// TIA Portal V20 program export: 1 tag tables, 1 data types, 3 data blocks, 8 code blocks (in call order from the OBs), 3 instance data blocks

VAR_GLOBAL   // PLC tag table "Default tag table"
   Tag_1 AT %M1.0 : Bool;
   Tag_2 AT %M10.0 : Bool;
   Tag_3 AT %M10.1 : Bool;
   Tag_4 AT %M10.2 : Bool;
   Tag_5 AT %M10.3 : Bool;
END_VAR

TYPE "F-link_UDT"
// stored: IsFailsafeCompliant true
   STRUCT
      ESTOP_OK : Bool;
      ESTOP_ack_req : Bool;
   END_STRUCT;
END_TYPE

DATA_BLOCK "Adatok_G2"   // DB2
{ S7_Optimized_Access := 'TRUE' }
// stored: MemoryReserve 100
BEGIN
END_DATA_BLOCK

DATA_BLOCK "Data_to_Safety"   // DB3
{ S7_Optimized_Access := 'TRUE' }
// stored: MemoryReserve 100
   VAR
      rcv_buffer : Array[0..121] of Byte;
      rcv_buffer2 : Array[0..121] of Byte;
   END_VAR
BEGIN
END_DATA_BLOCK

DATA_BLOCK "F-link_DB"   // DB2
{ S7_Optimized_Access := 'TRUE' }
// stored: MemoryReserve 100
   VAR
      receive : "F-link_UDT";
   END_VAR
BEGIN
END_DATA_BLOCK

ORGANIZATION_BLOCK "Main"   // OB1, LAD, ProgramCycle
TITLE = "Main Program Sweep (Cycle)"
{ S7_Optimized_Access := 'TRUE' }
// stored: SetENOAutomatically false
   VAR_INPUT
      Initial_Call : Bool;   // Initial call of this OB
      Remanence : Bool;   // =True, if remanent data are available
   END_VAR
BEGIN

REGION Network 1
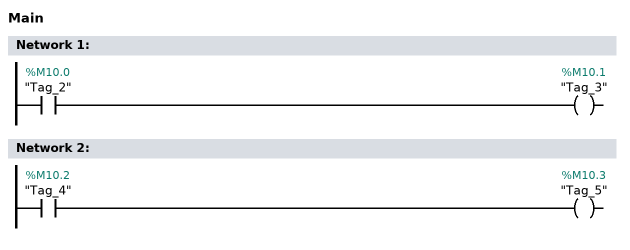
   RUNG wire#powerrail
      Contact( "Tag_2" )
      Coil( "Tag_3" )
   END_RUNG
   // the same network as SCL:
   "Tag_3" := "Tag_2";
END_REGION

REGION Network 2
   RUNG wire#powerrail
      Contact( "Tag_4" )
      Coil( "Tag_5" )
   END_RUNG
   // the same network as SCL:
   "Tag_5" := "Tag_4";
END_REGION
END_ORGANIZATION_BLOCK

ORGANIZATION_BLOCK "CyclicInterrupt"   // OB30, LAD, CyclicInterrupt
{ S7_Optimized_Access := 'TRUE' }
// stored: SetENOAutomatically false
   VAR_INPUT
      Initial_Call : Bool;   // Initial call of this OB
      Event_Count : Int;   // Events discarded
   END_VAR
BEGIN

REGION Network 1
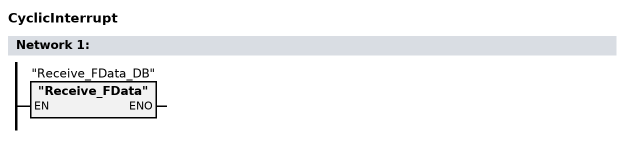
   RUNG wire#powerrail
      "Receive_FData_DB"()
   END_RUNG
   // the same network as SCL:
   "Receive_FData_DB"();   // "Receive_FData"
END_REGION
END_ORGANIZATION_BLOCK

FUNCTION_BLOCK "Receive_FData"   // FB2, FBD
{ S7_Optimized_Access := 'TRUE' }
// stored: MemoryReserve 100, SetENOAutomatically false
   VAR
      TRCV_Instance { S7_SetPoint := 'True'} : TRCV;
   END_VAR
BEGIN

REGION Network 1: ACK tömb fogadása
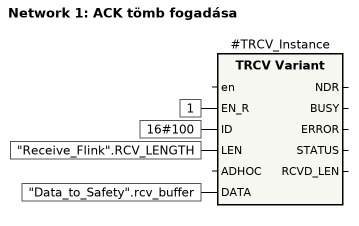
   #TRCV_Instance(EN_R := 1,   // TRCV
                  ID := 16#100,
                  LEN := "Receive_Flink".RCV_LENGTH,
                  DATA := "Data_to_Safety".rcv_buffer);
END_REGION
END_FUNCTION_BLOCK

FUNCTION_BLOCK "Main_Safety_RTG1"   // FB1, F_FBD
{ S7_Optimized_Access := 'TRUE' }
// stored: AutoNumber false
   VAR
      ESTOP1_Instance : ESTOP1;
   END_VAR
BEGIN

REGION Network 1
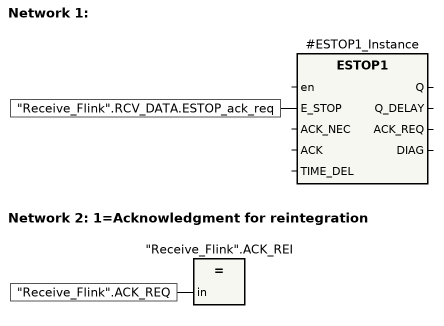
   #ESTOP1_Instance(E_STOP := "Receive_Flink".RCV_DATA.ESTOP_ack_req);   // ESTOP1
END_REGION

REGION Network 2: 1=Acknowledgment for reintegration
   "Receive_Flink".ACK_REI := "Receive_Flink".ACK_REQ;
END_REGION
END_FUNCTION_BLOCK

FUNCTION "PostProcess_Send" : Void   // FC2, FBD
{ S7_Optimized_Access := 'TRUE' }
// stored: SetENOAutomatically false
BEGIN

REGION Network 1
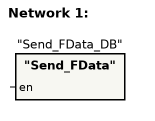
   "Send_FData_DB"();   // "Send_FData"
END_REGION
END_FUNCTION

FUNCTION_BLOCK "Send_FData"   // FB3, FBD
{ S7_Optimized_Access := 'TRUE' }
// stored: MemoryReserve 100, SetENOAutomatically false
   VAR
      TSEND_Instance { S7_SetPoint := 'True'} : TSEND;
      status_save { S7_SetPoint := 'True'} : Word;
      trigger : Bool;
   END_VAR
   VAR_TEMP   // added for the SCL form of the ladder/FBD networks
      _w1 : Bool;
   END_VAR
BEGIN

REGION Network 1
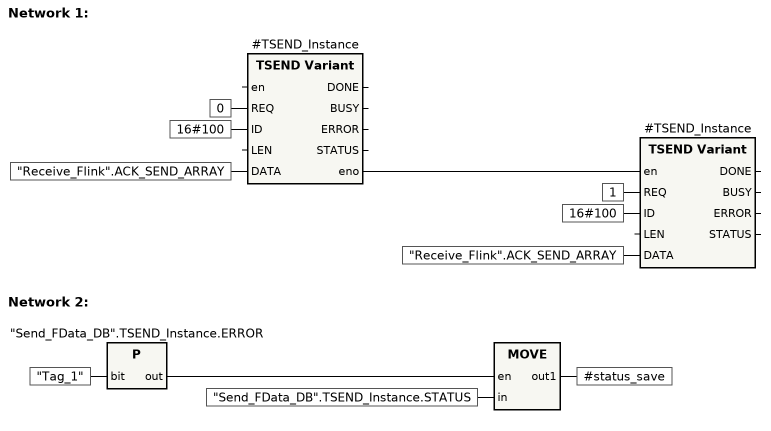
   #TSEND_Instance(REQ := 0, ID := 16#100, DATA := "Receive_Flink".ACK_SEND_ARRAY, ENO => #_w1);   // TSEND
   IF #_w1 THEN
       #TSEND_Instance(REQ := 1, ID := 16#100, DATA := "Receive_Flink".ACK_SEND_ARRAY);   // TSEND
   END_IF;
END_REGION

REGION Network 2
   #_w1 := "Send_FData_DB".TSEND_Instance.ERROR AND NOT "Tag_1";   // rising edge of "Send_FData_DB".TSEND_Instance.ERROR
   "Tag_1" := "Send_FData_DB".TSEND_Instance.ERROR;
   IF #_w1 THEN #status_save := "Send_FData_DB".TSEND_Instance.STATUS; END_IF;
END_REGION
END_FUNCTION_BLOCK

FUNCTION "PreProcess_Safety" : Void   // FC1, LAD
{ S7_Optimized_Access := 'TRUE' }
// stored: SetENOAutomatically false
BEGIN

REGION Network 1
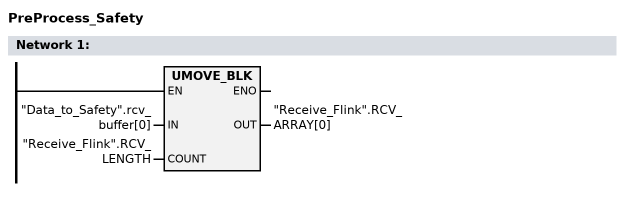
   UMOVE_BLK(IN := "Data_to_Safety".rcv_buffer[0],
             COUNT := "Receive_Flink".RCV_LENGTH,
             OUT => "Receive_Flink".RCV_ARRAY[0]);
END_REGION
END_FUNCTION

FUNCTION "Block_1" : Void
{ S7_Optimized_Access := 'TRUE' }
VERSION : 0.1

BEGIN
	(*
	Ez egy teszt feltoltés blokk
	*)
END_FUNCTION

DATA_BLOCK "Main_Safety_RTG1_DB"   // DB1, F_DB
NAME : FUSI
// stored: InstanceOfName Main_Safety_RTG1, InstanceOfType FB
"Main_Safety_RTG1"
BEGIN
END_DATA_BLOCK

DATA_BLOCK "Receive_FData_DB"   // DB4
// stored: InstanceOfName Receive_FData, InstanceOfType FB
"Receive_FData"
BEGIN
END_DATA_BLOCK

DATA_BLOCK "Send_FData_DB"   // DB5
// stored: InstanceOfName Send_FData, InstanceOfType FB
"Send_FData"
BEGIN
END_DATA_BLOCK
